{attribute addProperty BoxType "EL2262-0000-0004"}
{attribute addProperty Id "StartTimeNextOutputAT %I*StartTimeNextOutput_C2D377213240CycCount0AT %Q*CycCount0_307034DC1620Sample0AT %Q*ARRAY[0..9] OF Sample_ABF5BEA980100GapAT %Q*EMPTY_STRUCTURE000CycCount1AT %Q*CycCount1_7787FA1D1620Sample1AT %Q*ARRAY[0..9] OF Sample_4351E8AC80100Gap_1AT %Q*EMPTY_STRUCTURE000WcStateAT %I*WcState_F855686C1620InfoDataAT %I*InfoData_7231B2DD80100"}
{attribute addProperty CRC "693912799"}
{attribute addProperty SizeInBites "320"}
{attribute addProperty SizeInBytes "40"}
TYPE EL2262_CDC800E6 :
STRUCT
	{attribute addProperty Name "StartTimeNextOutput"}
	StartTimeNextOutput : StartTimeNextOutput_C2D37721;
	{attribute addProperty Name "CycCount0"}
	CycCount0 : CycCount0_307034DC;
	{attribute addProperty Name "Sample0"}
	Sample0 : ARRAY[0..9] OF Sample_ABF5BEA9;
	{attribute addProperty Name "Gap"}
	Gap : EMPTY_STRUCTURE;
	{attribute addProperty Name "CycCount1"}
	CycCount1 : CycCount1_7787FA1D;
	{attribute addProperty Name "Sample1"}
	Sample1 : ARRAY[0..9] OF Sample_4351E8AC;
	{attribute addProperty Name "Gap_1"}
	Gap_1 : EMPTY_STRUCTURE;
	{attribute addProperty Name "WcState"}
	WcState : WcState_F855686C;
	{attribute addProperty Name "InfoData"}
	InfoData : InfoData_7231B2DD;
END_STRUCT
END_TYPE

(* stored: Version 1.2.0.0, ProductVersion 3.1.4024.9
   DUT EL2262_CDC800E6: Id {b1c7eac6-7dc8-493c-a9fc-ae01711af6ca} *)
